Fanuc KAREL source: kt00042.KL

-- PROVISIONAL review KL for V770-1; original PC SHA256 e32519f1e061d2f207204dad9d13453661b2d362186f0c6fd23bfc2f034e62e5
-- Incomplete behavior may be omitted. Consult companion uncertainty JSON. Do not deploy.
PROGRAM KT00042
%NOLOCKGROUP
VAR
  R1 : REAL
  I2 : INTEGER
  OUT : REAL
BEGIN
  -- UNRESOLVED_PC offsets 5-16; opcodes 2E,23
  -- UNRESOLVED_PC offsets 21-32; opcodes 2E,23
  -- UNRESOLVED_PC offsets 37-57; opcodes 21,21,64,6A,23
  -- UNRESOLVED_PC offsets 62-66; opcodes 7F
END KT00042
